(* PLC project Main, Beckhoff Automation GmbH TwinCAT PLC Control 3.5.13.21 *)
(* stored: creationDateTime 2024-10-31T10:03:40.5522976, modificationDateTime 2024-10-31T10:03:40.5522976 *)

FUNCTION SquareSignal : REAL
VAR_INPUT
	ymin:				REAL; 	//Minimalwert
	ymax:				REAL; 	//Maximalwert
	w:					REAL; 	//Kreisfrequenz
	yoff:				REAL; 	//yoffset
	t : 				REAL;	//Zeit
END_VAR
VAR
	tempTime:			REAL;
	tempVar:			INT;
END_VAR

            tempTime := LMOD(lr_Value:=t,lr_Arg:=(2*PI)/w)/((2*PI)/w);

IF(tempTime >= (0.5)) THEN
	SquareSignal := ymax + yoff;
	RETURN;
ELSE
	SquareSignal := ymin + yoff;
	RETURN;
END_IF
          
END_FUNCTION
